FUNCTION_BLOCK FB_HwRefReactHeater EXTENDS FB_CanNodeBase
VAR_INPUT
END_VAR
VAR_OUTPUT
END_VAR
VAR
	//Eingänge
	nTempActual 	AT %I* : UINT;	//aktuelle Temperatur in 1/100tel °C 
	bTempCutoff 	AT %I* : BOOL;	//Übertemperaturabschaltung wurde aktiviert
	bVialDetected	AT %I* : BOOL;
	//Ausgänge
	nPidKp 			AT %Q* : UINT; 	//PID-Reglerparameter KP
	nPidKi 			AT %Q* : UINT;	//PID-Reglerparameter KI
	nPidKd 			AT %Q* : UINT;	//PID-Reglerparameter KD
	nPidTa 			AT %Q* : USINT;	//PID-Reglerparameter TA
	bHeatingOn		AT %Q* : BOOL;	//Heizer EIN
	nTempSetpoint	AT %Q* : USINT;	//Solltemperatur in °C (ohne Kommastellen)
	bResetVialDetect AT %Q* : BOOL;	//VialDetection zurücksetzen
END_VAR

IF bNodeEnabled THEN
	SUPER^();
END_IF

PROPERTY P_bHeatingOn : BOOL
SET
bHeatingOn := P_bHeatingOn;
END_SET
GET
P_bHeatingOn := bHeatingOn;
END_GET
END_PROPERTY

PROPERTY P_nTempActual : UINT
GET
P_nTempActual := nTempActual;
END_GET
END_PROPERTY

PROPERTY P_nPidKi : UINT
SET
nPidKi := P_nPidKi;
END_SET
GET
P_nPidKi := nPidKi;
END_GET
END_PROPERTY

PROPERTY P_nTempSetpoint : USINT
SET
nTempSetpoint := P_nTempSetpoint;
END_SET
GET
P_nTempSetpoint := nTempSetpoint;
END_GET
END_PROPERTY

PROPERTY P_nPidKd : UINT
GET
P_nPidKd := nPidKd;
END_GET
SET
nPidKd := P_nPidKd;
END_SET
END_PROPERTY

PROPERTY P_bResetVialDetect : BOOL
SET
bResetVialDetect := P_bResetVialDetect;
END_SET
GET
P_bResetVialDetect := bResetVialDetect;
END_GET
END_PROPERTY

PROPERTY P_nPidTa : USINT
GET
P_nPidTa := nPidTa;
END_GET
SET
nPidTa := P_nPidTa;
END_SET
END_PROPERTY

PROPERTY P_bTempCutoff : BOOL
GET
P_bTempCutoff := bTempCutoff;
END_GET
END_PROPERTY

PROPERTY P_nPidKp : UINT
GET
P_nPidKp := nPidKp;
END_GET
SET
nPidKp := P_nPidKp;
END_SET
END_PROPERTY

PROPERTY P_bVialDetected : BOOL
GET
P_bVialDetected := bVialDetected;
END_GET
END_PROPERTY

END_FUNCTION_BLOCK

(* stored: Version 1.1.0.1, ProductVersion 3.1.0.25
   POU FB_HwRefReactHeater: Id {5abe53b3-6214-4d33-9df7-cbf8b6449d94}
   Property P_bHeatingOn: Id {02ad8a62-217c-4a79-9dc6-11eb3f6b642e}
   Set Set: Id {0c138e36-c1a7-44f6-81ff-325fd48772e6}
   Get Get: Id {818e5d5b-db25-4cbd-83c8-6e8123bcaa09}
   Property P_nTempActual: Id {0f24e4e6-11ea-4524-ba63-8f5835318432}
   Get Get: Id {dbbfd260-b905-4d06-aca9-330784a9f0a1}
   Property P_nPidKi: Id {6a72c61d-eb3a-4897-9270-acfeb136317c}
   Set Set: Id {4cdf4e88-9447-43b6-9da7-97ec75670a09}
   Get Get: Id {cfad722f-bd78-4fb2-960c-09acb8da5e02}
   Property P_nTempSetpoint: Id {7ab31499-8a9d-4999-9de1-df2f92413df2}
   Set Set: Id {6c00b3d5-dbbb-4e27-9b7f-7f06a0eca952}
   Get Get: Id {8273363c-7450-451b-bd78-2af4241a0a24}
   Property P_nPidKd: Id {95261042-5ca6-43d1-8eaf-a50e3abae3b9}
   Get Get: Id {545aa0e0-6b59-4980-8ac7-876cffee93bb}
   Set Set: Id {7ed0762e-c99d-4df2-a01d-0baedbda3ae5}
   Property P_bResetVialDetect: Id {b849d57f-97f0-433f-921f-c4e47d98e54f}
   Set Set: Id {c7431377-78d8-4a0e-bd4b-447dca3c5ad6}
   Get Get: Id {d9d55842-6c99-4746-a5b5-55b43c0d7cc1}
   Property P_nPidTa: Id {c694ae83-4776-43f8-a7b9-ddc08d1571ba}
   Get Get: Id {7c213878-7c29-484c-af55-cc8718c8e652}
   Set Set: Id {890df8d9-42e2-4851-8de1-bd5ac1b8f1a0}
   Property P_bTempCutoff: Id {d9c1e38f-4977-49e4-addb-fa8b32805073}
   Get Get: Id {5f7db9fc-7ea1-4169-9dd3-03a9ee478b1f}
   Property P_nPidKp: Id {e3e215fb-5bd7-4c53-852e-3de57c46d95a}
   Get Get: Id {60a1ec41-622b-4aa6-97fe-c1772dd1c399}
   Set Set: Id {f922e583-2971-43b3-9566-a59278498722}
   Property P_bVialDetected: Id {fd7077fd-5e36-40f5-b713-a05700c2be82}
   Get Get: Id {8dc1b370-f910-4775-a923-c77ab9f8d10b} *)
